// ---- XTS_TRANSPORT/_Visualization/MOVER_VISU.TcVIS
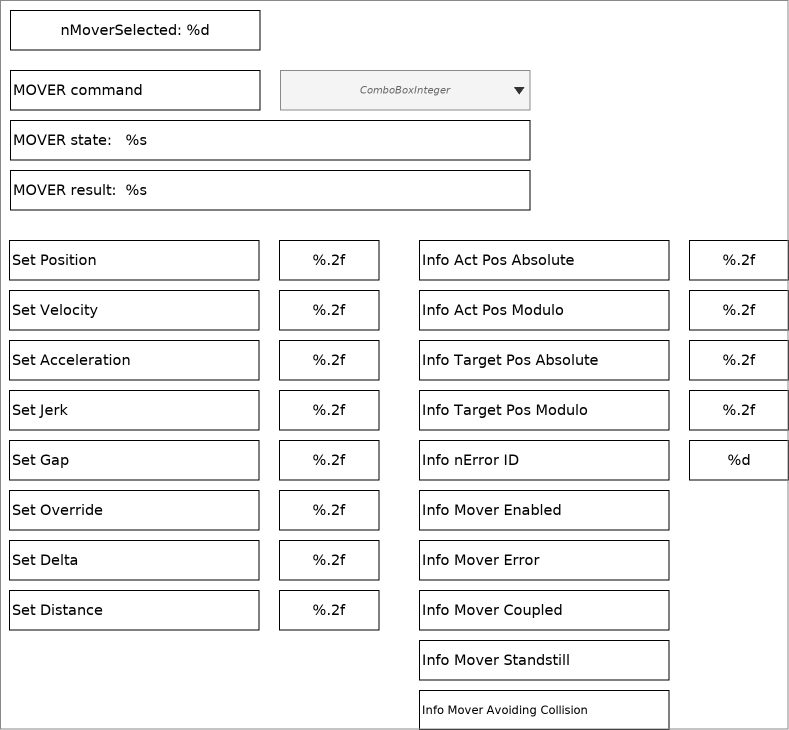
VISUALIZATION MOVER_VISU  // 789x730
    Rectangle (10,10 250x40), "nMoverSelected: %d", text variable: MAIN.nMoverSelected
        OnMouseClick: write the text variable via VisuDialogs.Numpad, min 1, max MAX_MOVER, title 'Selected Mover'
    Rectangle (10,120 520x40), "MOVER state: %s", text variable: MAIN.sMoverState
    Rectangle (10,70 250x40), "MOVER command"
    ComboBoxInteger (280,70 250x40), variable: GVL_XTS.MoverCtrl[MAIN.nMoverSelected].Cmd, text list: 'TL_E_CTRL_MOVER'
    Rectangle (10,170 520x40), "MOVER result: %s", text variable: MAIN.sMoverResult
    Rectangle (9,240 250x40), "Set Position"
    Rectangle (9,290 250x40), "Set Velocity"
    Rectangle (9,340 250x40), "Set Acceleration"
    Rectangle (9,390 250x40), "Set Jerk"
    Rectangle (9,440 250x40), "Set Gap"
    Rectangle (9,490 250x40), "Set Override"
    Rectangle (9,540 250x40), "Set Delta"
    Rectangle (9,590 250x40), "Set Distance"
    Rectangle (279,240 100x40), "%.2f", text variable: GVL_XTS.MoveData[MAIN.nMoverSelected].rPos
        OnMouseClick: write the text variable via Default
    Rectangle (279,290 100x40), "%.2f", text variable: GVL_XTS.MoveData[MAIN.nMoverSelected].rVelo
        OnMouseClick: write the text variable via Default
    Rectangle (279,340 100x40), "%.2f", text variable: GVL_XTS.MoveData[MAIN.nMoverSelected].rAcc
        OnMouseClick: write the text variable via Default
    Rectangle (279,390 100x40), "%.2f", text variable: GVL_XTS.MoveData[MAIN.nMoverSelected].rJerk
        OnMouseClick: write the text variable via Default
    Rectangle (279,440 100x40), "%.2f", text variable: GVL_XTS.MoveData[MAIN.nMoverSelected].rGap
        OnMouseClick: write the text variable via Default
    Rectangle (279,490 100x40), "%.2f", text variable: GVL_XTS.MoveData[MAIN.nMoverSelected].rOverride
        OnMouseClick: write the text variable via Default
    Rectangle (279,540 100x40), "%.2f", text variable: GVL_XTS.MoveData[MAIN.nMoverSelected].rDelta
        OnMouseClick: write the text variable via Default
    Rectangle (279,590 100x40), "%.2f", text variable: GVL_XTS.MoveData[MAIN.nMoverSelected].rDistance
        OnMouseClick: write the text variable via Default
    Rectangle (419,240 250x40), "Info Act Pos Absolute"
    Rectangle (419,290 250x40), "Info Act Pos Modulo"
    Rectangle (419,340 250x40), "Info Target Pos Absolute"
    Rectangle (419,390 250x40), "Info Target Pos Modulo"
    Rectangle (419,440 250x40), "Info nError ID"
    Rectangle (689,240 100x40), "%.2f", text variable: GVL_XTS.MoverInfo[MAIN.nMoverSelected].rAbsActPos
    Rectangle (689,290 100x40), "%.2f", text variable: GVL_XTS.MoverInfo[MAIN.nMoverSelected].rModuloActPos
    Rectangle (689,340 100x40), "%.2f", text variable: GVL_XTS.MoverInfo[MAIN.nMoverSelected].rAbsTargetPos
    Rectangle (689,390 100x40), "%.2f", text variable: GVL_XTS.MoverInfo[MAIN.nMoverSelected].rModuloTargetPos
    Rectangle (689,440 100x40), "%d", text variable: GVL_XTS.MoverInfo[MAIN.nMoverSelected].nErrorId
    Rectangle (419,490 250x40), "Info Mover Enabled", colour toggle: GVL_XTS.MoverInfo[MAIN.nMoverSelected].bMoverEnabled
    Rectangle (419,540 250x40), "Info Mover Error", colour toggle: GVL_XTS.MoverInfo[MAIN.nMoverSelected].bMoverError
    Rectangle (419,590 250x40), "Info Mover Coupled", colour toggle: GVL_XTS.MoverInfo[MAIN.nMoverSelected].bMoverCoupled
    Rectangle (419,640 250x40), "Info Mover Standstill", colour toggle: GVL_XTS.MoverInfo[MAIN.nMoverSelected].bMoverStandstill
    Rectangle (419,690 250x40), "Info Mover Avoiding Collision", colour toggle: GVL_XTS.MoverInfo[MAIN.nMoverSelected].bMoverAvoidingCollision
END_VISUALIZATION

// ---- XTS_TRANSPORT/_Visualization/SELECTOR_VISU.TcVIS
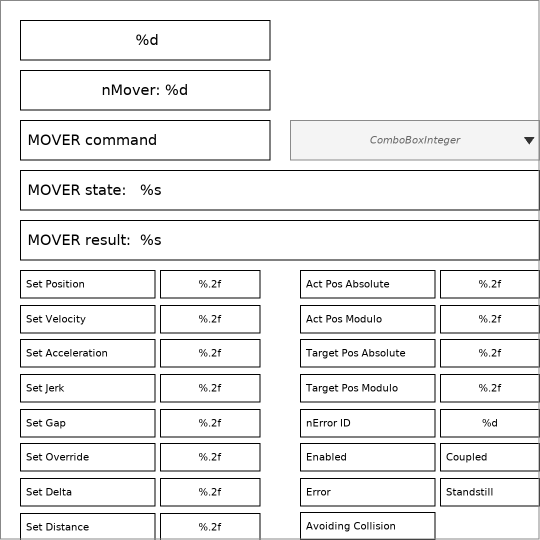
VISUALIZATION SELECTOR_VISU  // 540x540
    Frame (10,10 530x530)
        shows T_MOVER_SELECTOR(Control := GVL_XTS.SelectorCtrl, State := GVL_XTS.SelectorState, sState := MAIN.sSelectorState, sResult := MAIN.sSelectorResult)
END_VISUALIZATION

// ---- XTS_TRANSPORT/_Visualization/types/T_MOVER_SELECTOR.TcVIS
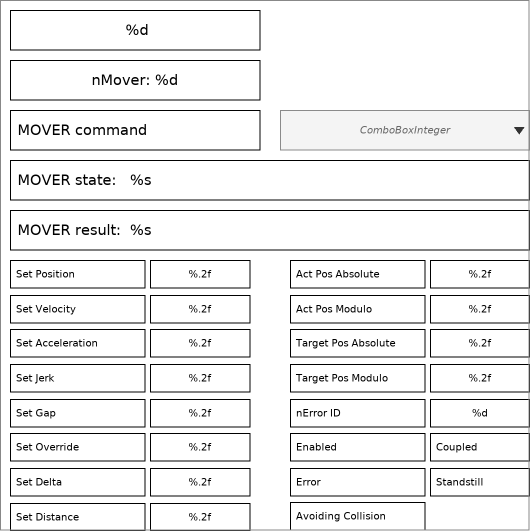
VISUALIZATION T_MOVER_SELECTOR  // 530x531
VAR_IN_OUT
	Control     : ST_MOVER_SELECTOR_CTRL;
  State       : ST_MOVER_SELECTOR_STATE;
  sState      : STRING;
  sResult     : STRING;
END_VAR
    Rectangle (10,60 250x40), "nMover: %d", text variable: Control.Mover
        OnMouseClick: write the text variable via VisuDialogs.Numpad, min 1, max MAX_MOVER, title 'Selected Mover'
    Rectangle (10,10 250x40), "%d", text variable: Control.Selector, text list: 'TL_E_MOVER_SELECTOR'
        OnMouseClick: write the text variable via VisuDialogs.Numpad, min 1, max MAX_MOVER, title 'Selected Mover'
    Rectangle (10,160 520x40), "MOVER state: %s", text variable: sState
    Rectangle (10,110 250x40), "MOVER command"
    ComboBoxInteger (280,110 250x40), variable: Control.Control.Cmd, text list: 'TL_E_CTRL_MOVER'
    Rectangle (10,210 520x40), "MOVER result: %s", text variable: sResult
    Rectangle (10,260 135x28), "Set Position"
    Rectangle (10,295 135x28), "Set Velocity"
    Rectangle (10,329 135x28), "Set Acceleration"
    Rectangle (10,364 135x28), "Set Jerk"
    Rectangle (10,399 135x28), "Set Gap"
    Rectangle (10,433 135x28), "Set Override"
    Rectangle (10,468 135x28), "Set Delta"
    Rectangle (10,503 135x28), "Set Distance"
    Rectangle (150,260 100x28), "%.2f", text variable: Control.Data.rPos
        OnMouseClick: write the text variable via Default
    Rectangle (150,295 100x28), "%.2f", text variable: Control.Data.rVelo
        OnMouseClick: write the text variable via Default
    Rectangle (150,329 100x28), "%.2f", text variable: Control.Data.rAcc
        OnMouseClick: write the text variable via Default
    Rectangle (150,364 100x28), "%.2f", text variable: Control.Data.rJerk
        OnMouseClick: write the text variable via Default
    Rectangle (150,399 100x28), "%.2f", text variable: Control.Data.rGap
        OnMouseClick: write the text variable via Default
    Rectangle (150,433 100x28), "%.2f", text variable: Control.Data.rOverride
        OnMouseClick: write the text variable via Default
    Rectangle (150,468 100x28), "%.2f", text variable: Control.Data.rDelta
        OnMouseClick: write the text variable via Default
    Rectangle (150,503 100x28), "%.2f", text variable: Control.Data.rDistance
        OnMouseClick: write the text variable via Default
    Rectangle (290,260 135x28), "Act Pos Absolute"
    Rectangle (290,295 135x28), "Act Pos Modulo"
    Rectangle (290,329 135x28), "Target Pos Absolute"
    Rectangle (290,364 135x28), "Target Pos Modulo"
    Rectangle (290,399 135x28), "nError ID"
    Rectangle (430,260 100x28), "%.2f", text variable: GVL_XTS.MoverInfo[MAIN.nMoverSelected].rAbsActPos
    Rectangle (430,295 100x28), "%.2f", text variable: GVL_XTS.MoverInfo[MAIN.nMoverSelected].rModuloActPos
    Rectangle (430,329 100x28), "%.2f", text variable: GVL_XTS.MoverInfo[MAIN.nMoverSelected].rAbsTargetPos
    Rectangle (430,364 100x28), "%.2f", text variable: GVL_XTS.MoverInfo[MAIN.nMoverSelected].rModuloTargetPos
    Rectangle (430,399 100x28), "%d", text variable: GVL_XTS.MoverInfo[MAIN.nMoverSelected].nErrorId
    Rectangle (290,433 135x28), "Enabled", colour toggle: GVL_XTS.MoverInfo[MAIN.nMoverSelected].bMoverEnabled
    Rectangle (290,468 135x28), "Error", colour toggle: GVL_XTS.MoverInfo[MAIN.nMoverSelected].bMoverError
    Rectangle (430,433 100x28), "Coupled", colour toggle: GVL_XTS.MoverInfo[MAIN.nMoverSelected].bMoverCoupled
    Rectangle (430,468 100x28), "Standstill", colour toggle: GVL_XTS.MoverInfo[MAIN.nMoverSelected].bMoverStandstill
    Rectangle (290,502 135x28), "Avoiding Collision", colour toggle: GVL_XTS.MoverInfo[MAIN.nMoverSelected].bMoverAvoidingCollision
END_VISUALIZATION
